{attribute 'GeneratedUsingTerminal: EK1100-0000-0018'}
{attribute addProperty BoxType "EK1100-0000-0018"}
{attribute addProperty Id "Beckhoff_EPP4xxxEK1122Beckhoff_EPP4xxxEK1122_A3CF6D4E166"}
{attribute addProperty CRC "2265388989"}
{attribute addProperty Size "166"}
TYPE Beckhoff_EPP4xxx_870717BD EXTENDS EK1100_1FC0878B :
STRUCT
	{attribute addProperty Name "Beckhoff_EPP4xxxEK1122"}
	{attribute addProperty PreviousPort "Beckhoff EPP4xxx : B"}
	Beckhoff_EPP4xxxEK1122 : Beckhoff_EPP4xxxEK1122_A3CF6D4E;
END_STRUCT
END_TYPE

(* stored: Version 1.2.0.0, ProductVersion 3.1.4024.9
   DUT Beckhoff_EPP4xxx_870717BD: Id {bf01b973-6ed4-4e50-94b6-ef298f131ddf} *)
